// TIA Portal V20 export
DATA_BLOCK "instTeachingPosMendrelAnodeFrontAxisZ"   // DB468
// stored: InstanceOfName LER_TeachingPos_Interface, InstanceOfType FB
"LER_TeachingPos_Interface"
   // VAR_INPUT
   //    enable : Bool;
   //    selectTeachingPos : SInt;
   //    indexTeachingPos : SInt;
   // END_VAR
   // VAR_IN_OUT
   //    configurationSetPositions : Array[0..15] of "LBC_typeAxis64PosSetPosition";
   //    moduleInterface : "LBC_typeAxis64PosInterface";
   //    hmiInterface : Array[0..48] of "LER_TypeTeachingPosInterface";
   // END_VAR
   // VAR
   //    statPulse : Array[0..9] of Bool;
   //    statTonTimer : Array[0..15] of TON_TIME;
   //    statLastTeachingPosIndex : SInt;
   // END_VAR
BEGIN
END_DATA_BLOCK
